(* IEC 61131-3 sources: repolevel_ST_code_completion/output/0122完整版本_无planner目前sota/repoeval_Interation_HowTo/readful_result_no_provide, 2 files *)

(* ---- FirstPublish.st ---- *)
VAR
    publisher: MQTT.MQTTPublish;
    doPublish: BOOL;
    init: BOOL;
    sendPayload: STRING := 'testPayload';
END_VAR

IF NOT init THEN
    init := TRUE;
    publisher.SetMqttInOut(MQTT_IN_OUT := HowTo.MQTT_IN_OUT);
END_IF

publisher(
    Topic := ADR('TestTopic/FromCodesys'),
    PayloadString := ADR(sendPayload),
    PublishAsString := TRUE,
    QoSIn := MQTT.QoS.ExactlyOnce,
    MRetain := FALSE,
    send := doPublish);
END_FUNCTION_BLOCK

(* ---- FirstSubscription.st ---- *)
VAR
    collector: MQTT.CallbackCollector;
    SUB1: MQTT.MQTTSubscribe;
    init: BOOL := FALSE;
    receiver: MQTT.ReceiveString;
END_VAR

IF NOT init THEN
    init := TRUE;
    SUB1.SetMqttInOut(MQTT_IN_OUT := HowTo.MQTT_IN_OUT);
    collector.put(instance := receiver);
    receiver.initAsFindTopic(compString := ADR('TestTopic/FromCodesys'), returnHit := TRUE);
END_IF

SUB1(
    Subscribe := TRUE,
    Topic := ADR('TestTopic/FromCodesys'),
    QoSSubscribe := MQTT.QoS.ExactlyOnce,
    ExpectingString := TRUE,
    Callback := collector);
END_FUNCTION_BLOCK
